Staubli VAL3: wizard.pgx

public program wizard()
  local num l_nSelect
  local bool l_bSelect
begin
  l_nSelect=0
  cls()
  while l_nSelect<3
    switch l_nSelect
      case 0
        call use:typeMenu(8,">>")
        call use:typeMenu(7,"<<")
        gotoxy(1,1)
        put("1")
        do
          nPage=getKey()
          if(nPage==278)
            l_nSelect=l_nSelect+1
            l_bSelect=true
          elseIf(nPage==277)
            l_nSelect=5
            return
          endIf
        until l_bSelect==true
      break
      case 1
        call use:typeMenu(8,">>")
        call use:typeMenu(7,"<<")
        gotoxy(1,1)
        put("2")
        do
          nPage=getKey()
          if(nPage==278)
            l_nSelect=l_nSelect+1
            l_bSelect=true
          elseIf(nPage==277)
            l_nSelect=l_nSelect-1
            l_bSelect=true
          endIf
        until l_bSelect==true
      break
      case 2
        call use:typeMenu(8,">>")
        call use:typeMenu(7,"<<")
        gotoxy(1,1)
        put("3")
        do
          nPage=getKey()
          if(nPage==278)
            l_nSelect=l_nSelect+1
            l_bSelect=true
          elseIf(nPage==277)
            l_nSelect=l_nSelect-1
            l_bSelect=true
          endIf
        until l_bSelect==true
      break
      case 3
      break
      case 4
      break
    endSwitch
  endWhile
end
